(* IEC 61131-3 sources: openplc-temperature-control/plc/boolean_test/pous/programs, 1 file *)

(* ---- main.st ---- *)
PROGRAM main
  VAR
    TestInput : BOOL := FALSE;
    Enable : BOOL := TRUE;
    TestOutput : BOOL := FALSE;
  END_VAR

TestOutput := TestInput AND Enable;

END_PROGRAM
